Fanuc KAREL source: kt00476.KL

-- PROVISIONAL review KL for V770-1; original PC SHA256 bde5f7a5bf2be6b9bf287b62811c36c2079432a1398173d905ae5572b67b48fb
-- Incomplete behavior may be omitted. Consult companion uncertainty JSON. Do not deploy.
PROGRAM KT00476
%NOLOCKGROUP
-- UNRESOLVED_DECL P1 type=000101
-- UNRESOLVED_DECL P2 type=000101
-- UNRESOLVED_DECL OUT type=000106
BEGIN
  -- UNRESOLVED_PC offsets 5-34; opcodes 49,49,60,7E,4A
  -- UNRESOLVED_PC offsets 39-43; opcodes 7F
END KT00476
